% RSLogix 500 project Star Delta.RSS, saved by version 8.10.00.18 %
PROJECT "UNTITLED"    % processor: type code 162 %

PROGRAM FILES
  LAD 2   2 rungs

DATA FILES
  S2 STATUS  83 elements
  B3 BINARY  1 elements
  T4 TIMER  1 elements
  C5 COUNTER  1 elements
  R6 CONTROL  1 elements
  N7 INTEGER  1 elements
  F8 FLOAT  1 elements

LADDER 2
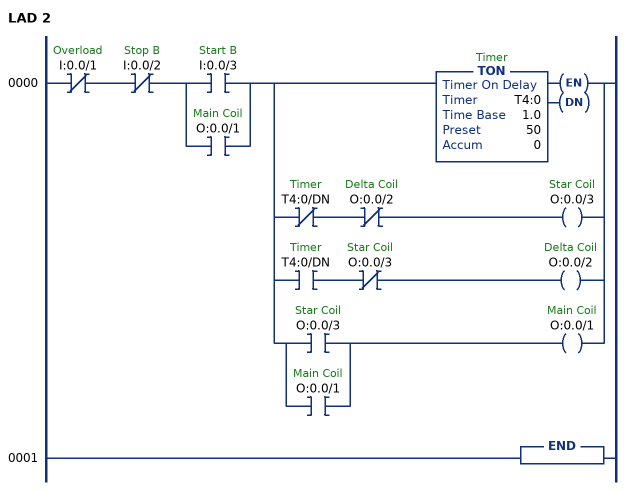
% Rung: 0 %  % edit flag set %
SOR XIO I:0.0/1 XIO I:0.0/2 BST XIC I:0.0/3 NXB XIC O:0.0/1 BND BST TON T4:0 1.0 50 0 NXB XIO T4:0/DN XIO O:0.0/2 OTE O:0.0/3 NXB XIC T4:0/DN XIO O:0.0/3 OTE O:0.0/2 NXB BST XIC O:0.0/3 NXB XIC O:0.0/1 BND OTE O:0.0/1 BND EOR
%   I:0.0/1  "Overload" %
%   I:0.0/2  "Stop B" %
%   I:0.0/3  "Start B" %
%   O:0.0/1  "Main Coil" %
%   T4:0  "Timer" %
%   O:0.0/2  "Delta Coil" %
%   O:0.0/3  "Star Coil" %
% Rung: 1 %
SOR END EOR
